{attribute 'qualified_only'}
{attribute 'strict'}
TYPE EChamberMode :
(
	Unknown := 0,
	Maintenance,
	Run
);
END_TYPE

(* stored: Version 1.1.0.1, ProductVersion 3.1.4024.12
   DUT EChamberMode: Id {ac8a4ad6-2ebb-4628-969f-6dd0dd65cebb} *)
